(* CODESYS project MQTT2.ecp

Project tree, tasks and I/O mapping:
  Controller : 750-8202 PFC200 2ETH RS, WAGO, order no. 0750-8202, version 5.15.4.20
    application Application
      libraries: ; WagoAppJSON, 1.1.0.11 (WAGO); WagoAppCloud, * (WAGO); WagoAppTime, 1.7.3.3 (WAGO)
      task PLC_Task (cyclic, interval 100 ms, priority 15) calls PLC_PRG
      program PLC_PRG [ST]
      global variables GVL_MQTT
      Lysstyring/
        program PRG_Lys_Innelys [ST]
        program PRG_Lys_Utelys_Normal [ST]
        program PRG_Lys_Utelys_Nattslukk [ST]
        program PRG_Lys [ST]
      FB&DT/
        data type dtShelly1
        function block fbShelly1_Publish [ST]
        function block fbShelly1_Subscribe [ST]
      MQTT/
        program PRG_Publish1 [ST]
        program PRG_Subscribe [ST]
        program PRG_Status [ST]
        program PRG_Publish [ST]
        program PRG_MQTT [ST]
    Kbus : Kbus, WAGO, version 1.4.0.2
        unmapped channels: K-BUS diagnostics
    MODBUS
      MODBUS : MODBUS, WAGO, order no. n/a, version 1.1.1.15
        LocalDeviceModbus : MODBUS Slave, WAGO, order no. n/a, version 1.1.1.15
            settings: OffsetMap = 0
            input  MbMqttTopicPart : WORD  // 
          TcpSettings : Modbus TCP Slave, WAGO, order no. n/a, version 1.1.1.15
              settings: TCP connection watchdog = 200 10ms
    Serial
      COM1 : COM1, WAGO, version 0.0.0.19
  Generic_MODBUS_Master : ThirdParty Modbus Master, WAGO, order no. GenericModbusMaster, version 1.0.0.1
*)

// Controller/Application/FB&DT/dtShelly1
TYPE dtShelly1 :
STRUCT
	
	sTopic: STRING;
	sState: STRING;
	sCommand: STRING;
	sLastCommand: STRING;

END_STRUCT
END_TYPE

// Controller/Application/GVL_MQTT
VAR_GLOBAL
	
//Felles
	tTid: TOD;
//2019
	SE2019WR002: dtShelly1:=(sTopic:= '943B25');
	SE2019WR003: dtShelly1:=(sTopic:= '554056');;
	SE2019WR004: dtShelly1:=(sTopic:= '553D87');;
	SE2019WR006: dtShelly1:=(sTopic:= '55E599');;
	SE2019WR012: dtShelly1:=(sTopic:= 'B8D834');;
	SE2019WR013: dtShelly1:=(sTopic:= 'B8DD56');;
	SE2019WR014: dtShelly1:=(sTopic:= 'B8D53D');;
	SE2019WR015: dtShelly1:=(sTopic:= 'B8EB06');;
	SE2019WR016: dtShelly1:=(sTopic:= 'B8D9EB');;
	SE2019WR017: dtShelly1:=(sTopic:= 'B8D985');;
	SE2019WR018: dtShelly1:=(sTopic:= 'B8DA02');;
	SE2019WR019: dtShelly1:=(sTopic:= 'B8CA18');;

//2020	
	SE2020WR001: dtShelly1:=(sTopic:= '045CE8');;
	SE2020WR002: dtShelly1:=(sTopic:= '05284A');;
	SE2020WR003: dtShelly1:=(sTopic:= '053424');;
	SE2020WR004: dtShelly1:=(sTopic:= '044B19');;
	SE2020WR005: dtShelly1:=(sTopic:= '04B587');;
	SE2020WR006: dtShelly1:=(sTopic:= '04E727');;
	SE2020WR007: dtShelly1:=(sTopic:= '04D932');;
	
//2021
	SE2021WR001: dtShelly1:=(sTopic:= '8CAAB5');;
	SE2021WR002: dtShelly1:=(sTopic:= '8CAAB561B879');;
	SE2021WR003: dtShelly1:=(sTopic:= '8CAAB55E0512');;
	SE2021WR007: dtShelly1:=(sTopic:= '8CAAB55E0576');;
	SE2021WR009: dtShelly1:=(sTopic:= '8CAAB561554E');;
	SE2021WR017: dtShelly1:=(sTopic:= '8CAAB55D9602');;
	
END_VAR

// Controller/Application/PLC_PRG
PROGRAM PLC_PRG
VAR
	
	

END_VAR

PRG_MQTT();
PRG_Lys();

END_PROGRAM

// Controller/Application/MQTT/PRG_MQTT
PROGRAM PRG_MQTT
VAR
END_VAR

PRG_Status();
PRG_Subscribe();
PRG_Publish();

END_PROGRAM

// Controller/Application/MQTT/PRG_Status
PROGRAM PRG_Status
VAR
	
	oFbStatus 			: WagoAppCloud.FbStatus_NativeMQTT;
	xMyError			: BOOL := FALSE;
	xConnectedToMyCloud	: BOOL := FALSE;
	rMyFillLevel		: REAL := 0;
	uliMyOutgoingBlocks	: ULINT := 0;
	
END_VAR

oFbStatus(xEnabled := TRUE,
		   xError => xMyError,
		   xCloudConnected => xConnectedToMyCloud,			// Will be FALSE after network timeout occured 
		   rCacheFillLevel => rMyFillLevel,					// Increasing value indicates bad network or overload
		   uliOutgoingDataBlocks => uliMyOutgoingBlocks);

END_PROGRAM

// Controller/Application/MQTT/PRG_Subscribe
PROGRAM PRG_Subscribe
VAR
	
	Subscribe		: fbShelly1_Subscribe;
	Subscribe1		: fbShelly1_Subscribe;
	Subscribe2		: fbShelly1_Subscribe;
	Subscribe3		: fbShelly1_Subscribe;
	Subscribe4		: fbShelly1_Subscribe;
	Subscribe5		: fbShelly1_Subscribe;
	Subscribe6		: fbShelly1_Subscribe;
	Subscribe7		: fbShelly1_Subscribe;
	Subscribe8		: fbShelly1_Subscribe;
	Subscribe9		: fbShelly1_Subscribe;
	Subscribe10		: fbShelly1_Subscribe;
	Subscribe11		: fbShelly1_Subscribe;
	Subscribe12		: fbShelly1_Subscribe;
	Subscribe13		: fbShelly1_Subscribe;
	Subscribe14		: fbShelly1_Subscribe;
	Subscribe15		: fbShelly1_Subscribe;
	Subscribe16		: fbShelly1_Subscribe;
	Subscribe17		: fbShelly1_Subscribe;
	Subscribe18		: fbShelly1_Subscribe;
	Subscribe19		: fbShelly1_Subscribe;
	Subscribe20		: fbShelly1_Subscribe;
	Subscribe21		: fbShelly1_Subscribe;
	Subscribe22		: fbShelly1_Subscribe;
	Subscribe23		: fbShelly1_Subscribe;
	Subscribe24		: fbShelly1_Subscribe;
	
END_VAR

Subscribe		(sSubTopic:= SE2019WR002.sTopic, 	sState=> SE2019WR002.sState);
Subscribe1		(sSubTopic:= SE2019WR003.sTopic, 	sState=> SE2019WR003.sState);
Subscribe2		(sSubTopic:= SE2019WR004.sTopic, 	sState=> SE2019WR004.sState);
Subscribe3		(sSubTopic:= SE2019WR006.sTopic, 	sState=> SE2019WR006.sState);
Subscribe4		(sSubTopic:= SE2019WR012.sTopic, 	sState=> SE2019WR012.sState);
Subscribe5		(sSubTopic:= SE2019WR013.sTopic, 	sState=> SE2019WR013.sState);
Subscribe6		(sSubTopic:= SE2019WR014.sTopic, 	sState=> SE2019WR014.sState);
Subscribe7		(sSubTopic:= SE2019WR015.sTopic, 	sState=> SE2019WR015.sState);
Subscribe8		(sSubTopic:= SE2019WR016.sTopic, 	sState=> SE2019WR016.sState);
Subscribe9		(sSubTopic:= SE2019WR017.sTopic, 	sState=> SE2019WR017.sState);
Subscribe10		(sSubTopic:= SE2019WR018.sTopic, 	sState=> SE2019WR018.sState);
Subscribe11		(sSubTopic:= SE2019WR019.sTopic, 	sState=> SE2019WR019.sState);
Subscribe12		(sSubTopic:= SE2020WR001.sTopic, 	sState=> SE2020WR001.sState);
Subscribe13		(sSubTopic:= SE2020WR002.sTopic, 	sState=> SE2020WR002.sState);
Subscribe14		(sSubTopic:= SE2020WR003.sTopic, 	sState=> SE2020WR003.sState);
Subscribe15		(sSubTopic:= SE2020WR004.sTopic, 	sState=> SE2020WR004.sState);
Subscribe16		(sSubTopic:= SE2020WR005.sTopic, 	sState=> SE2020WR005.sState);
Subscribe17		(sSubTopic:= SE2020WR006.sTopic, 	sState=> SE2020WR006.sState);
Subscribe18		(sSubTopic:= SE2020WR007.sTopic, 	sState=> SE2020WR007.sState);
Subscribe19		(sSubTopic:= SE2021WR001.sTopic, 	sState=> SE2021WR001.sState);
Subscribe20		(sSubTopic:= SE2021WR002.sTopic, 	sState=> SE2021WR002.sState);
Subscribe21		(sSubTopic:= SE2021WR003.sTopic, 	sState=> SE2021WR003.sState);
Subscribe22		(sSubTopic:= SE2021WR007.sTopic, 	sState=> SE2021WR007.sState);
Subscribe23		(sSubTopic:= SE2021WR009.sTopic, 	sState=> SE2021WR009.sState);
Subscribe24		(sSubTopic:= SE2021WR017.sTopic, 	sState=> SE2021WR017.sState);

END_PROGRAM

// Controller/Application/FB&DT/fbShelly1_Subscribe
FUNCTION_BLOCK fbShelly1_Subscribe
VAR_INPUT
	
	sSubTopic		: STRING(255);

END_VAR
VAR_OUTPUT
	
	sState			: STRING(255);
	
END_VAR
VAR
	
	oFbSubscribe 		: WagoAppCloud.FbSubscribeMQTT;
	aSubscriptionData	: ARRAY [0..254] OF BYTE;
	
END_VAR

sSubTopic:= CONCAT('shellies/shelly1-', sSubTopic );
sSubTopic:= CONCAT(sSubTopic, '/relay/0');

IoConfig_Globals_Mapping.MbMqttTopicPart;
oFbSubscribe(xSubscribe := TRUE, sTopic := sSubTopic, eQoS := eQualityOfService.QoS0, aPayloadData:= aSubscriptionData);
MemCopySecure(pDest:= ADR(sState), udiDestSize:= 255, pSource:= ADR(aSubscriptionData), udiSourceSize:= oFbSubscribe.dwRxNBytes, bPadding:= 0);

END_FUNCTION_BLOCK

// Controller/Application/MQTT/PRG_Publish
PROGRAM PRG_Publish
VAR
	
	Publish: fbShelly1_Publish;
	i: INT:= 0;

END_VAR

CASE i OF
	0:
		Publish(sPubTopic:= SE2019WR002.sTopic, sStatus:= SE2019WR002.sState, sCommand:= SE2019WR002.sCommand, sLastCommandIn:= SE2019WR002.sLastCommand , sLastCommandOut=> SE2019WR002.sLastCommand);
		i:= i+1;
		RETURN;
	1:
		Publish(sPubTopic:= SE2019WR003.sTopic, sStatus:= SE2019WR003.sState, sCommand:= SE2019WR003.sCommand, sLastCommandIn:= SE2019WR003.sLastCommand , sLastCommandOut=> SE2019WR003.sLastCommand);
		i:= i+1;
		RETURN;
	2:
		Publish(sPubTopic:= SE2019WR004.sTopic, sStatus:= SE2019WR004.sState, sCommand:= SE2019WR004.sCommand, sLastCommandIn:= SE2019WR004.sLastCommand , sLastCommandOut=> SE2019WR004.sLastCommand);
		i:= i+1;
		RETURN;
	3:
		Publish(sPubTopic:= SE2019WR006.sTopic, sStatus:= SE2019WR006.sState, sCommand:= SE2019WR006.sCommand, sLastCommandIn:= SE2019WR006.sLastCommand , sLastCommandOut=> SE2019WR006.sLastCommand);
		i:= i+1;
		RETURN;
	4:
		Publish(sPubTopic:= SE2019WR012.sTopic, sStatus:= SE2019WR012.sState, sCommand:= SE2019WR012.sCommand, sLastCommandIn:= SE2019WR012.sLastCommand , sLastCommandOut=> SE2019WR012.sLastCommand);
		i:= i+1;
		RETURN;
	5:
		Publish(sPubTopic:= SE2019WR013.sTopic, sStatus:= SE2019WR013.sState, sCommand:= SE2019WR013.sCommand, sLastCommandIn:= SE2019WR013.sLastCommand , sLastCommandOut=> SE2019WR013.sLastCommand);
		i:= i+1;
		RETURN;
	6:
		Publish(sPubTopic:= SE2019WR014.sTopic, sStatus:= SE2019WR014.sState, sCommand:= SE2019WR014.sCommand, sLastCommandIn:= SE2019WR014.sLastCommand , sLastCommandOut=> SE2019WR014.sLastCommand);
		i:= i+1;
		RETURN;
	7:
		Publish(sPubTopic:= SE2019WR015.sTopic, sStatus:= SE2019WR015.sState, sCommand:= SE2019WR015.sCommand, sLastCommandIn:= SE2019WR015.sLastCommand , sLastCommandOut=> SE2019WR015.sLastCommand);
		i:= i+1;
		RETURN;
	8:
		Publish(sPubTopic:= SE2019WR016.sTopic, sStatus:= SE2019WR016.sState, sCommand:= SE2019WR016.sCommand, sLastCommandIn:= SE2019WR016.sLastCommand , sLastCommandOut=> SE2019WR016.sLastCommand);
		i:= i+1;
		RETURN;
	9:
		Publish(sPubTopic:= SE2019WR017.sTopic, sStatus:= SE2019WR017.sState, sCommand:= SE2019WR017.sCommand, sLastCommandIn:= SE2019WR017.sLastCommand , sLastCommandOut=> SE2019WR017.sLastCommand);
		i:= i+1;
		RETURN;
	10:
		Publish(sPubTopic:= SE2019WR018.sTopic, sStatus:= SE2019WR018.sState, sCommand:= SE2019WR018.sCommand, sLastCommandIn:= SE2019WR018.sLastCommand , sLastCommandOut=> SE2019WR018.sLastCommand);
		i:= i+1;
		RETURN;
	11:
		Publish(sPubTopic:= SE2019WR019.sTopic, sStatus:= SE2019WR019.sState, sCommand:= SE2019WR019.sCommand, sLastCommandIn:= SE2019WR019.sLastCommand , sLastCommandOut=> SE2019WR019.sLastCommand);
		i:= i+1;
		RETURN;
	12:
		Publish(sPubTopic:= SE2020WR001.sTopic, sStatus:= SE2020WR001.sState, sCommand:= SE2020WR001.sCommand, sLastCommandIn:= SE2020WR001.sLastCommand , sLastCommandOut=> SE2020WR001.sLastCommand);
		i:= i+1;
		RETURN;
	13:
		Publish(sPubTopic:= SE2020WR002.sTopic, sStatus:= SE2020WR002.sState, sCommand:= SE2020WR002.sCommand, sLastCommandIn:= SE2020WR002.sLastCommand , sLastCommandOut=> SE2020WR002.sLastCommand);
		i:= i+1;
		RETURN;
	14:
		Publish(sPubTopic:= SE2020WR003.sTopic, sStatus:= SE2020WR003.sState, sCommand:= SE2020WR003.sCommand, sLastCommandIn:= SE2020WR003.sLastCommand , sLastCommandOut=> SE2020WR003.sLastCommand);
		i:= i+1;
		RETURN;
	15:	
		Publish(sPubTopic:= SE2020WR004.sTopic, sStatus:= SE2020WR004.sState, sCommand:= SE2020WR004.sCommand, sLastCommandIn:= SE2020WR004.sLastCommand , sLastCommandOut=> SE2020WR004.sLastCommand);
		i:= i+1;
		RETURN;
	16:	
		Publish(sPubTopic:= SE2020WR005.sTopic, sStatus:= SE2020WR005.sState, sCommand:= SE2020WR005.sCommand, sLastCommandIn:= SE2020WR005.sLastCommand , sLastCommandOut=> SE2020WR005.sLastCommand);
		i:= i+1;
		RETURN;
	17:	
		Publish(sPubTopic:= SE2020WR006.sTopic, sStatus:= SE2020WR006.sState, sCommand:= SE2020WR006.sCommand, sLastCommandIn:= SE2020WR006.sLastCommand , sLastCommandOut=> SE2020WR006.sLastCommand);
		i:= i+1;
		RETURN;
	18:	
		Publish(sPubTopic:= SE2020WR007.sTopic, sStatus:= SE2020WR007.sState, sCommand:= SE2020WR007.sCommand, sLastCommandIn:= SE2020WR007.sLastCommand , sLastCommandOut=> SE2020WR007.sLastCommand);
		i:= i+1;
		RETURN;
	19:	
		Publish(sPubTopic:= SE2021WR001.sTopic, sStatus:= SE2021WR001.sState, sCommand:= SE2021WR001.sCommand, sLastCommandIn:= SE2021WR001.sLastCommand , sLastCommandOut=> SE2021WR001.sLastCommand);
		i:= i+1;
		RETURN;
	20:	
		Publish(sPubTopic:= SE2021WR002.sTopic, sStatus:= SE2021WR002.sState, sCommand:= SE2021WR002.sCommand, sLastCommandIn:= SE2021WR002.sLastCommand , sLastCommandOut=> SE2021WR002.sLastCommand);
		i:= i+1;
		RETURN;
	21:	
		Publish(sPubTopic:= SE2021WR003.sTopic, sStatus:= SE2021WR003.sState, sCommand:= SE2021WR003.sCommand, sLastCommandIn:= SE2021WR003.sLastCommand , sLastCommandOut=> SE2021WR003.sLastCommand);
		i:= i+1;
		RETURN;
	22:
		Publish(sPubTopic:= SE2021WR007.sTopic, sStatus:= SE2021WR007.sState, sCommand:= SE2021WR007.sCommand, sLastCommandIn:= SE2021WR007.sLastCommand , sLastCommandOut=> SE2021WR007.sLastCommand);
		i:= i+1;
		RETURN;
	23:	
		Publish(sPubTopic:= SE2021WR009.sTopic, sStatus:= SE2021WR009.sState, sCommand:= SE2021WR009.sCommand, sLastCommandIn:= SE2021WR009.sLastCommand , sLastCommandOut=> SE2021WR009.sLastCommand);
		i:= i+1;
		RETURN;
	24:	
		Publish(sPubTopic:= SE2021WR017.sTopic, sStatus:= SE2021WR017.sState, sCommand:= SE2021WR017.sCommand, sLastCommandIn:= SE2021WR017.sLastCommand , sLastCommandOut=> SE2021WR017.sLastCommand);
		i:= 0;
END_CASE

END_PROGRAM

// Controller/Application/FB&DT/fbShelly1_Publish
FUNCTION_BLOCK fbShelly1_Publish
VAR_INPUT
	sPubTopic		: STRING(255);
	sStatus			: STRING(255);
	sCommand 		: STRING(255);
	sLastCommandIn	: STRING(255);
END_VAR
VAR_OUTPUT
	
	sLastCommandOut	: STRING(255);

END_VAR
VAR
	
	aBuffer			: ARRAY[0..255] OF BYTE;
	dwBytesCount 	: DWORD;
	fbPublish 		: WagoAppCloud.FbPublishMQTT:=(eQualityOfService := eQualityOfService.QoS0);
	xTrigger		: BOOL := TRUE;
	
END_VAR

sPubTopic:= CONCAT('shellies/shelly1-', sPubTopic);
sPubTopic:= CONCAT(sPubTopic,  '/relay/0/command');

IF sCommand <> sLastCommandIn AND NOT fbPublish.xBusy THEN
//Copy JSON to buffer
	dwBytesCount := Length(sCommand);
	MemCopy(pDest := ADR(aBuffer), pSource := ADR(sCommand), udiSize := dwBytesCount);

//Trigger the transmission
	xTrigger := TRUE;
	
//Lagrer forgje command
	sLastCommandOut:= sCommand;
ELSIF NOT fbPublish.xBusy THEN
	sLastCommandOut:= sCommand;
END_IF

fbPublish(	sTopic := sPubTopic, dwSize := dwBytesCount, aData := aBuffer, xTrigger := xTrigger);

END_FUNCTION_BLOCK

// Controller/Application/Lysstyring/PRG_Lys
PROGRAM PRG_Lys
VAR
END_VAR

tTid:= DT_TO_TOD(FuGetLocalDateAndTime());
PRG_Lys_Innelys();
PRG_Lys_Utelys_Nattslukk();
PRG_Lys_Utelys_Normal();

END_PROGRAM

// Controller/Application/Lysstyring/PRG_Lys_Innelys
PROGRAM PRG_Lys_Innelys
VAR

	xIndoor: BOOL;
	xIndoor_Force: BOOL;
	tIndoorOn: TOD:= TOD#06:00:00;
	tIndoorOff: TOD:= TOD#21:00:00;
	
END_VAR

//Indoor
	IF tTid = tIndoorOn OR xIndoor_Force THEN
		xIndoor:= TRUE;
	ELSIF tTid = tIndoorOff THEN
		xIndoor:= FALSE;
	END_IF

//Setter alle relee til rett verdi
	IF xIndoor THEN
		SE2020WR001.sCommand:= 'on';
		SE2020WR002.sCommand:= 'on';
		SE2020WR003.sCommand:= 'on';
		SE2020WR004.sCommand:= 'on';
		SE2020WR005.sCommand:= 'on';
		SE2020WR006.sCommand:= 'on';
		SE2020WR007.sCommand:= 'on';
		SE2021WR001.sCommand:= 'on';
		SE2021WR002.sCommand:= 'on';
		SE2021WR003.sCommand:= 'on';
		SE2021WR009.sCommand:= 'on';
	ELSE
		SE2020WR001.sCommand:= 'off';
		SE2020WR002.sCommand:= 'off';
		SE2020WR003.sCommand:= 'off';
		SE2020WR004.sCommand:= 'off';
		SE2020WR005.sCommand:= 'off';
		SE2020WR006.sCommand:= 'off';
		SE2020WR007.sCommand:= 'off';
		SE2021WR001.sCommand:= 'off';
		SE2021WR002.sCommand:= 'off';
		SE2021WR003.sCommand:= 'off';
		SE2021WR009.sCommand:= 'off';
	END_IF
	
	(*
//Trigger ny sending hvis status ikke stemmer med ønsket verdi
	IF SE2020WR001.sCommand <> SE2020WR001.sState THEN
		SE2020WR001.sLastCommand:= '';
	END_IF
	IF SE2020WR002.sCommand <> SE2020WR002.sState THEN
		SE2020WR002.sLastCommand:= '';
	END_IF
	IF SE2020WR003.sCommand <> SE2020WR003.sState THEN
		SE2020WR003.sLastCommand:= '';
	END_IF
	IF SE2020WR004.sCommand <> SE2020WR004.sState THEN
		SE2020WR004.sLastCommand:= '';
	END_IF
	IF SE2020WR005.sCommand <> SE2020WR005.sState THEN
		SE2020WR005.sLastCommand:= '';
	END_IF
	IF SE2020WR006.sCommand <> SE2020WR006.sState THEN
		SE2020WR006.sLastCommand:= '';
	END_IF
	IF SE2020WR007.sCommand <> SE2020WR007.sState THEN
		SE2020WR007.sLastCommand:= '';
	END_IF
	IF SE2021WR001.sCommand <> SE2021WR001.sState THEN
		SE2021WR001.sLastCommand:= '';
	END_IF
	IF SE2021WR002.sCommand <> SE2021WR002.sState THEN
		SE2021WR002.sLastCommand:= '';
	END_IF
	IF SE2021WR003.sCommand <> SE2021WR003.sState THEN
		SE2021WR003.sLastCommand:= '';
	END_IF
	IF SE2021WR009.sCommand <> SE2021WR009.sState THEN
		SE2021WR009.sLastCommand:= '';
	END_IF
	*)

END_PROGRAM

// Controller/Application/Lysstyring/PRG_Lys_Utelys_Nattslukk
PROGRAM PRG_Lys_Utelys_Nattslukk
VAR
	
	xOutdoorOffNight: BOOL;	
	xOutdoorOffNight_Force: BOOL;
	tOutdoorOffNightOn_1: TOD:= TOD#06:00:00;
	tOutdoorOffNightOff_1: TOD:= TOD#09:00:00;
	tOutdoorOffNightOn_2: TOD:= TOD#18:00:00;
	tOutdoorOffNightOff_2: TOD:= TOD#21:00:00;

END_VAR

//OutdoorOffNight Tidsstyring
	IF tTid = tOutdoorOffNightOn_1 OR tTid = tOutdoorOffNightOn_2 OR xOutdoorOffNight_Force THEN
		xOutdoorOffNight:= TRUE;
	ELSIF tTid = tOutdoorOffNightOff_1 OR tTid = tOutdoorOffNightOff_2 THEN
		xOutdoorOffNight:= FALSE;
	END_IF

//Setter alle relee til rett verdi
	IF xOutdoorOffNight THEN
		SE2019WR002.sCommand:= 'on';
		SE2019WR003.sCommand:= 'on';
		SE2019WR004.sCommand:= 'on';
		SE2019WR006.sCommand:= 'on';
		SE2019WR013.sCommand:= 'on';
		SE2019WR014.sCommand:= 'on';
	ELSE
		SE2019WR002.sCommand:= 'off';
		SE2019WR003.sCommand:= 'off';
		SE2019WR004.sCommand:= 'off';
		SE2019WR006.sCommand:= 'off';
		SE2019WR013.sCommand:= 'off';
		SE2019WR014.sCommand:= 'off';
	END_IF
	
(*
//Trigger ny sending hvis status ikke stemmer med ønsket verdi
	IF SE2019WR002.sCommand <> SE2019WR002.sState THEN
		SE2019WR002.sLastCommand:= '';
	END_IF
	IF SE2019WR003.sCommand <> SE2019WR003.sState THEN
		SE2019WR003.sLastCommand:= '';
	END_IF
	IF SE2019WR004.sCommand <> SE2019WR004.sState THEN
		SE2019WR004.sLastCommand:= '';
	END_IF
	IF SE2019WR006.sCommand <> SE2019WR006.sState THEN
		SE2019WR006.sLastCommand:= '';
	END_IF
	IF SE2019WR013.sCommand <> SE2019WR013.sState THEN
		SE2019WR013.sLastCommand:= '';
	END_IF
	IF SE2019WR014.sCommand <> SE2019WR014.sState THEN
		SE2019WR014.sLastCommand:= '';
	END_IF
	*)

END_PROGRAM

// Controller/Application/Lysstyring/PRG_Lys_Utelys_Normal
PROGRAM PRG_Lys_Utelys_Normal
VAR

	xOutdoorNormal: BOOL;
	xOutdoorNormal_Force: BOOL;
	tOutdoorNormalOn: TOD:= TOD#20:00:00;
	tOutdoorNormalOff: TOD:= TOD#06:00:00;

END_VAR

//OutdoorNormal
	IF tTid = tOutdoorNormalOn OR xOutdoorNormal_Force THEN
		xOutdoorNormal:= TRUE;
	ELSIF tTid = tOutdoorNormalOff THEN
		xOutdoorNormal:= FALSE;
	END_IF

//Setter alle relee til rett verdi
	IF xOutdoorNormal THEN
		GVL_MQTT.SE2019WR012.sCommand:= 'on';
		GVL_MQTT.SE2019WR015.sCommand:= 'on';
		GVL_MQTT.SE2019WR016.sCommand:= 'on';
		GVL_MQTT.SE2019WR017.sCommand:= 'on';
		GVL_MQTT.SE2019WR018.sCommand:= 'on';
		GVL_MQTT.SE2019WR019.sCommand:= 'on';
		GVL_MQTT.SE2021WR007.sCommand:= 'on';
		GVL_MQTT.SE2021WR017.sCommand:= 'on';
	ELSE
		GVL_MQTT.SE2019WR012.sCommand:= 'off';
		GVL_MQTT.SE2019WR015.sCommand:= 'off';
		GVL_MQTT.SE2019WR016.sCommand:= 'off';
		GVL_MQTT.SE2019WR017.sCommand:= 'off';
		GVL_MQTT.SE2019WR018.sCommand:= 'off';
		GVL_MQTT.SE2019WR019.sCommand:= 'off';
		GVL_MQTT.SE2021WR007.sCommand:= 'off';
		GVL_MQTT.SE2021WR017.sCommand:= 'off';
	END_IF
	
(*
//Trigger ny sending hvis status ikke stemmer med ønsket verdi
	IF SE2019WR012.sCommand <> SE2019WR012.sState THEN
		SE2019WR012.sLastCommand:= '';
	END_IF
	IF SE2019WR015.sCommand <> SE2019WR015.sState THEN
		SE2019WR015.sLastCommand:= '';
	END_IF
	IF SE2019WR016.sCommand <> SE2019WR016.sState THEN
		SE2019WR016.sLastCommand:= '';
	END_IF
	IF SE2019WR017.sCommand <> SE2019WR017.sState THEN
		SE2019WR017.sLastCommand:= '';
	END_IF
	IF SE2019WR018.sCommand <> SE2019WR018.sState THEN
		SE2019WR018.sLastCommand:= '';
	END_IF
	IF SE2019WR019.sCommand <> SE2019WR019.sState THEN
		SE2019WR019.sLastCommand:= '';
	END_IF
	IF SE2021WR007.sCommand <> SE2021WR007.sState THEN
		SE2021WR007.sLastCommand:= '';
	END_IF
	IF SE2021WR017.sCommand <> SE2021WR017.sState THEN
		SE2021WR017.sLastCommand:= '';
	END_IF
	*)

END_PROGRAM

// Controller/Application/MQTT/PRG_Publish1
PROGRAM PRG_Publish1
VAR
	
	Publish: fbPublish;
	Publish1: fbPublish;
	Publish2: fbPublish;
	Publish3: fbPublish;
	Publish4: fbPublish;
	Publish5: fbPublish;
	Publish6: fbPublish;
	Publish7: fbPublish;
	Publish8: fbPublish;
	Publish9: fbPublish;
	Publish10: fbPublish;
	Publish11: fbPublish;
	Publish12: fbPublish;
	Publish13: fbPublish;
	Publish14: fbPublish;
	Publish15: fbPublish;
	Publish16: fbPublish;
	Publish17: fbPublish;
	Publish18: fbPublish;
	Publish19: fbPublish;
	Publish20: fbPublish;
	Publish21: fbPublish;
	Publish22: fbPublish;
	Publish23: fbPublish;
	Publish24: fbPublish;
	
	test: STRING;
	test1: STRING;
	i: INT:= 0;

END_VAR


		Publish(sPubTopic:= SE2019WR002.sTopic, sCommand:= SE2019WR002.sCommand, sLastCommandIn:= SE2019WR002.sLastCommand , sLastCommandOut=> SE2019WR002.sLastCommand);

		Publish1(sPubTopic:= SE2019WR003.sTopic, sCommand:= SE2019WR003.sCommand, sLastCommandIn:= SE2019WR003.sLastCommand , sLastCommandOut=> SE2019WR003.sLastCommand);

		Publish2(sPubTopic:= SE2019WR004.sTopic, sCommand:= SE2019WR004.sCommand, sLastCommandIn:= SE2019WR004.sLastCommand , sLastCommandOut=> SE2019WR004.sLastCommand);

		Publish3(sPubTopic:= SE2019WR006.sTopic, sCommand:= SE2019WR006.sCommand, sLastCommandIn:= SE2019WR006.sLastCommand , sLastCommandOut=> SE2019WR006.sLastCommand);

		Publish4(sPubTopic:= SE2019WR012.sTopic, sCommand:= SE2019WR012.sCommand, sLastCommandIn:= SE2019WR012.sLastCommand , sLastCommandOut=> SE2019WR012.sLastCommand);

		Publish5(sPubTopic:= SE2019WR013.sTopic, sCommand:= SE2019WR013.sCommand, sLastCommandIn:= SE2019WR013.sLastCommand , sLastCommandOut=> SE2019WR013.sLastCommand);

		Publish6(sPubTopic:= SE2019WR014.sTopic, sCommand:= SE2019WR014.sCommand, sLastCommandIn:= SE2019WR014.sLastCommand , sLastCommandOut=> SE2019WR014.sLastCommand);

		Publish7(sPubTopic:= SE2019WR015.sTopic, sCommand:= SE2019WR015.sCommand, sLastCommandIn:= SE2019WR015.sLastCommand , sLastCommandOut=> SE2019WR015.sLastCommand);

		Publish8(sPubTopic:= SE2019WR016.sTopic, sCommand:= SE2019WR016.sCommand, sLastCommandIn:= SE2019WR016.sLastCommand , sLastCommandOut=> SE2019WR016.sLastCommand);

		Publish9(sPubTopic:= SE2019WR017.sTopic, sCommand:= SE2019WR017.sCommand, sLastCommandIn:= SE2019WR017.sLastCommand , sLastCommandOut=> SE2019WR017.sLastCommand);

		Publish10(sPubTopic:= SE2019WR018.sTopic, sCommand:= SE2019WR018.sCommand, sLastCommandIn:= SE2019WR018.sLastCommand , sLastCommandOut=> SE2019WR018.sLastCommand);

		Publish11(sPubTopic:= SE2019WR019.sTopic, sCommand:= SE2019WR019.sCommand, sLastCommandIn:= SE2019WR019.sLastCommand , sLastCommandOut=> SE2019WR019.sLastCommand);

		Publish12(sPubTopic:= SE2020WR001.sTopic, sCommand:= SE2020WR001.sCommand, sLastCommandIn:= SE2020WR001.sLastCommand , sLastCommandOut=> SE2020WR001.sLastCommand);

		Publish13(sPubTopic:= SE2020WR002.sTopic, sCommand:= SE2020WR002.sCommand, sLastCommandIn:= SE2020WR002.sLastCommand , sLastCommandOut=> SE2020WR002.sLastCommand);

		Publish14(sPubTopic:= SE2020WR003.sTopic, sCommand:= SE2020WR003.sCommand, sLastCommandIn:= SE2020WR003.sLastCommand , sLastCommandOut=> SE2020WR003.sLastCommand);

		Publish15(sPubTopic:= SE2020WR004.sTopic, sCommand:= SE2020WR004.sCommand, sLastCommandIn:= SE2020WR004.sLastCommand , sLastCommandOut=> SE2020WR004.sLastCommand);
	
		Publish16(sPubTopic:= SE2020WR005.sTopic, sCommand:= SE2020WR005.sCommand, sLastCommandIn:= SE2020WR005.sLastCommand , sLastCommandOut=> SE2020WR005.sLastCommand);

		Publish17(sPubTopic:= SE2020WR006.sTopic, sCommand:= SE2020WR006.sCommand, sLastCommandIn:= SE2020WR006.sLastCommand , sLastCommandOut=> SE2020WR006.sLastCommand);
	
		Publish18(sPubTopic:= SE2020WR007.sTopic, sCommand:= SE2020WR007.sCommand, sLastCommandIn:= SE2020WR007.sLastCommand , sLastCommandOut=> SE2020WR007.sLastCommand);

		Publish19(sPubTopic:= SE2021WR001.sTopic, sCommand:= SE2021WR001.sCommand, sLastCommandIn:= SE2021WR001.sLastCommand , sLastCommandOut=> SE2021WR001.sLastCommand);

		Publish20(sPubTopic:= SE2021WR002.sTopic, sCommand:= SE2021WR002.sCommand, sLastCommandIn:= SE2021WR002.sLastCommand , sLastCommandOut=> SE2021WR002.sLastCommand);

		Publish21(sPubTopic:= SE2021WR003.sTopic, sCommand:= SE2021WR003.sCommand, sLastCommandIn:= SE2021WR003.sLastCommand , sLastCommandOut=> SE2021WR003.sLastCommand);

		Publish22(sPubTopic:= SE2021WR007.sTopic, sCommand:= SE2021WR007.sCommand, sLastCommandIn:= SE2021WR007.sLastCommand , sLastCommandOut=> SE2021WR007.sLastCommand);

		Publish23(sPubTopic:= SE2021WR009.sTopic, sCommand:= SE2021WR009.sCommand, sLastCommandIn:= SE2021WR009.sLastCommand , sLastCommandOut=> SE2021WR009.sLastCommand);

		Publish24(sPubTopic:= SE2021WR017.sTopic, sCommand:= SE2021WR017.sCommand, sLastCommandIn:= SE2021WR017.sLastCommand , sLastCommandOut=> SE2021WR017.sLastCommand);

END_PROGRAM
